{attribute 'qualified_only'}
{attribute 'strict'}
TYPE E_ProcessState :
(
	None := 0,
	Active,
	Finish,
	NG
);
END_TYPE

(* stored: Version 1.1.0.1, ProductVersion 3.1.4024.10
   DUT E_ProcessState: Id {e5d8179d-1003-45a9-8bed-32df42c5efed} *)
